Staubli VAL3: start.pgx

public program start()
  local string l_sConnect
begin

  //初始化Wacoh Force/Torque Sensor
  call initSensor("io:Wacoh",l_sConnect)
  if l_sConnect=="yes"
    putln("Connection success!")
    delay(1.0)
  else
    putln("Connection fail!")
    delay(1.0)
  endIf

  //创建同步任务，循环获取传感器的Force/Torque数据（采集频率0.004s，频率为250Hz，可设置调节，超时是否需打开？）
  taskCreateSync "getForces",0.004,bOverRun,loopReadForce()

  //创建异步任务，将采集的传感器数据发送至用户界面实时显示
  taskCreate "user",20,userInterface()

end
